// TIA Portal V20 program export: 1 tag tables, 0 data types, 0 data blocks, 3 code blocks (in call order from the OBs), 0 instance data blocks

VAR_GLOBAL   // PLC tag table "Default tag table"
   adat1 AT %IW0 : Int;
   adat2 AT %IW2 : Int;
   adat3 AT %IW4 : Int;
   adat4 AT %IW6 : Int;
   adat5 AT %IW8 : Int;
   adat6 AT %IW10 : Int;
   adat7 AT %IW12 : Int;
   adat8 AT %IW14 : Word;
END_VAR

ORGANIZATION_BLOCK "Main"   // OB1, LAD, ProgramCycle
TITLE = "Main Program Sweep (Cycle)"
{ S7_Optimized_Access := 'TRUE' }
// stored: SetENOAutomatically false
   VAR_INPUT
      Initial_Call : Bool;   // Initial call of this OB
      Remanence : Bool;   // =True, if remanent data are available
   END_VAR
BEGIN

REGION Network 1
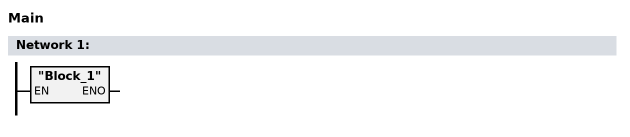
   RUNG wire#powerrail
      "Block_1"()
   END_RUNG
   // the same network as SCL:
   "Block_1"();
END_REGION
END_ORGANIZATION_BLOCK

FUNCTION "Block_1" : Void   // FC1, FBD
{ S7_Optimized_Access := 'TRUE' }
// stored: SetENOAutomatically false
BEGIN
END_FUNCTION

FUNCTION "Block_2" : Void   // FC2, FBD
{ S7_Optimized_Access := 'TRUE' }
// stored: SetENOAutomatically false
BEGIN
END_FUNCTION
